TYPE udtEthercatSlaveStatus :
STRUCT
	Address : WORD;
	Name : STRING[31];
	DeviceState: BYTE;
	LinkState: BYTE;
	SlaveStateBits: ST_EcSlaveStateBits;
END_STRUCT
END_TYPE

(* stored: Version 1.1.0.1, ProductVersion 3.1.4020.12
   DUT udtEthercatSlaveStatus: Id {82058017-8533-40c9-a236-124677e7aee0} *)
